// TIA Portal V16 export
// export: Created 2022-01-20T18:36:29.2285565Z, ExportSetting WithDefaults, DisplayName Totally Integrated Automation Portal, DisplayVersion V16, DisplayName TIA Portal Version Control Interface, DisplayVersion V16, DisplayName TIA Portal Openness, DisplayVersion V16, DisplayName STEP 7 Professional, DisplayVersion V16, DisplayName STEP 7 Safety, DisplayVersion V16, DisplayName WinCC Advanced, DisplayVersion V16
DATA_BLOCK "TCPIP_COMMS_DB"   // DB1
VERSION : 0.1
// stored: AutoNumber true, InstanceOfName TCPIP_COMMS, InstanceOfType FB
"TCPIP_COMMS"
   // VAR
   //    TCON : Struct
   //       REQ : Bool;
   //       DONE : Bool;
   //       BUSY : Bool;
   //       ERROR : Bool;
   //       STATUS : UInt;
   //       DONESAVE : Bool;
   //    END_STRUCT;
   //    TDISCON : Struct
   //       REQ : Bool;
   //       DONE : Bool;
   //       BUSY : Bool;
   //       ERROR : Bool;
   //       DONESAVE : Bool;
   //       STATUS : UInt;
   //    END_STRUCT;
   //    TSEND : Struct
   //       REQ : Bool;
   //       DONE : Bool;
   //       BUSY : Bool;
   //       ERROR : Bool;
   //       DONESAVE : Bool;
   //       STATUS : UInt;
   //    END_STRUCT;
   //    TRCV : Struct
   //       EN_R : Bool;
   //       NDR : Bool;
   //       BUSY : Bool;
   //       ERROR : Bool;
   //       STATUS : UInt;
   //       RCVD_LEN : UDInt;
   //    END_STRUCT;
   //    ReceivedString : String;
   //    TCON_DB { ExternalAccessible := 'False'; ExternalVisible := 'False'; ExternalWritable := 'False'} : TCON;
   //    TDISCON_DB { ExternalAccessible := 'False'; ExternalVisible := 'False'; ExternalWritable := 'False'} : TDISCON;
   //    TSEND_DB { ExternalAccessible := 'False'; ExternalVisible := 'False'; ExternalWritable := 'False'} : TSEND;
   //    TRCV_DB { ExternalAccessible := 'False'; ExternalVisible := 'False'; ExternalWritable := 'False'} : TRCV;
   // END_VAR
BEGIN
END_DATA_BLOCK
